FUNCTION TryConvert_DINT_TO_LWORD : BOOL
VAR_INPUT
	in : DINT;
	out : REFERENCE TO LWORD;
END_VAR

IF in < DatatypeLimits.MIN_VALUE_OF_DINT_WHICH_CAN_BE_HELD_IN_A_LWORD THEN
	RETURN;
END_IF

out := DINT_TO_LWORD(in);
TryConvert_DINT_TO_LWORD := TRUE;

END_FUNCTION

(* stored: Version 1.1.0.1, ProductVersion 3.1.4024.12
   POU TryConvert_DINT_TO_LWORD: Id {e3ff2489-b091-4b8c-81ed-1d7e86ccd467}, SpecialFunc None *)
